// TIA Portal V16 export
// export: Created 2021-05-25T16:14:41.9140055Z, ExportSetting WithDefaults, DisplayName Totally Integrated Automation Portal, DisplayVersion V16, DisplayName TIA Portal Version Control Interface, DisplayVersion V16, DisplayName TIA Portal Openness, DisplayVersion V16, DisplayName STEP 7 Professional, DisplayVersion V16, DisplayName STEP 7 Safety, DisplayVersion V16, DisplayName WinCC Unified SCADA Engineering System, DisplayVersion V16
DATA_BLOCK "dbSystemParam"   // DB320
{ S7_Optimized_Access := 'TRUE'; DB_Accessible_From_OPC_UA := 'FALSE' }
VERSION : 0.1
// stored: AutoNumber false, DBAccessibleFromOPCUA false
   VAR RETAIN
      KONCNA_POZICIJA_VIJACENJA_DES_NAZAJ_FilterTime : USInt := 10;
      KONCNA_POZICIJA_VIJACENJA_DES_NAPREJ_FilterTime : USInt := 10;
      KONCNA_POZICIJA_VIJACENJA_LEVO_NAZAJ_FilterTime : USInt := 12;
      KONCNA_POZICIJA_VIJACENJA_LEVO_NAPREJ_FilterTime : USInt := 15;
      DlyTimeToStart_TRAK_VIJAC : Int := 5;
      DlyTimeToStop_TRAK_VIJAC : Int := 1;
      DlyTimeToStart_VIBRO : Int := 5;
      DlyTimeToStop_VIBRO : Int := 15;
      StandbyTimeTrakaVijac : UDInt := 15;
      DlyTimeForAlarmAddNewHelix : UInt := 10;
   END_VAR
BEGIN
END_DATA_BLOCK
